// TIA Portal V17 export
// export: Created 2024-10-17T14:16:17.8144427Z, ExportSetting WithDefaults, DisplayName Totally Integrated Automation Portal, DisplayVersion V17 Update 4, DisplayName TIA Portal Openness, DisplayVersion V17 Update 4, DisplayName TIA Portal Version Control Interface, DisplayVersion V17, DisplayName SINAMICS Startdrive Advanced, DisplayVersion V17 Update2, DisplayName SINAMICS Startdrive G130, G150, S120, S150, SINAMICS MV, S210, DisplayVersion V17 Update2, DisplayName SINAMICS Startdrive G110M, G120, G120C, G120D, G120P, G115D, DisplayVersion V17 Update2, DisplayName STEP 7 Professional, DisplayVersion V17 Update 4, DisplayName STEP 7 Safety, DisplayVersion V17, DisplayName WinCC Advanced / Unified PC, DisplayVersion V17 Update 4
TYPE "LPMLV2022_typeModeStateTimes"
TITLE = LPMLV2022_typeModeStateTimes
// Support: tech.team.motioncontrol@siemens.com
// stored: IsFailsafeCompliant false
   STRUCT
      Mode { ExternalWritable := 'False'} : DInt;   // Mode Time Values for each Mode. This tag represents the cumulative amount of time (in seconds) spent in each Mode since the last timer and counter reset was executed
      State { ExternalWritable := 'False'} : Array[0.."LPMLV2022_ADMIN_NUMBER_OF_STATES_UPPER_LIM"] of DInt;   // State Time Values for each State in each Mode. This tag represents the cumulative amount of time (in seconds) spent in each state of a particular Mode since the last timer and counter reset was executed
   END_STRUCT;
END_TYPE
